# B&R Automation Studio project SuperTrak_Distribution
Automation Studio 4.12.5.95 SP; Demo project with Standard control, Axis coupling and Anti-Sloshing; technology packages: mapp 5.20.0, mappMotion 5.20.2, mappView 5.20.0

## Configuration APC910

CPU 5PC900.TS17-00, AutomationRuntime E4.91, Build 4.1.2, Safety 0.0, Vc V4.34.2

### Task classes (Cpu.sw)
```
Cyclic#1 (cycle 800 us, tolerance 0 us):
  ST_Main <- Source.SuperTrak.ST_Main.prg
  ST_Logic <- Source.SuperTrak.ST_Logic.prg
  ST_Visu <- Source.SuperTrak.ST_Visu.prg
  AxisCtrl <- Source.Axis.AxisCtrl.prg
DataObjects: McAcpSys, Acp10sys
NcDataObjects: McDriveLog
Binaries: STComTexts, McAcpDrv, udbdef, McAcpSim, mvLoader, arflatprv, McProfGen, TCLang, TCData, arcoal, arsvcreg, iomap, asfw, Config_3, Role, ashwac, sysconf, Config_2, arconfig, Config_1, TC, ashwd, Config, User, acp10cfg, Acp10map1, Acp10map, AxisConfig, OpcUaMap
Libraries: operator, AsBrMath, asstring, MpAlarmX, MpServer, McBase, MpBase, McAxis, McPureVAx, MpAxis, McAcpPar, HmiSupport, runtime, astime, AsIecCon, AsBrStr, standard, ArEventLog, AsArLog, sys_lib, McAcpAx, AsTCP, FileIO, AsIOTime, AsUDP, AsETH, AsARCfg, brsystem, AsGuard, AsHttp, AsXml, AsIOAcc, AsArSdm, AsIODiag, AsIO, AsIOMMan, DataObj, AsArProf, SuperTrak, aspciext, arssl, powerlnk, asepl, aruser, DevDetect, LogHelper, StCom
```

### Hardware
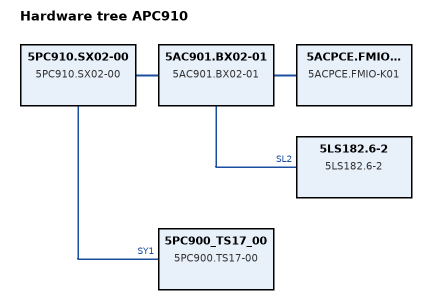
```
5AC901.BX02-01 : 5AC901.BX02-01 v1.1.1.0  [SY -> 5PC910.SX02-00.SY3]
5ACPCE.FMIO-K01 : 5ACPCE.FMIO-K01 v1.0.6.0  [SL -> 5AC901.BX02-01.SL1]
5LS182.6-2 : 5LS182.6-2 v1.9.0.0  [SL -> 5AC901.BX02-01.SL2]
  Connector IF1:
    DNAConfiguration = manual
    CycleTime = 800
5PC900_TS17_00 : 5PC900.TS17-00 v2.1.0.0  [SY -> 5PC910.SX02-00.SY1]
  ConfigurationID = SuperTrak_DistributionPackage
  UserPartitionSize = 100
  Simulation = 1
  VolatileGlobalPvSize = 262144
  TimerDeviceType = EPLX2X
  TimerDevice = 5LS182.6-2.IF1
  TaskClassIdleTime = 800
  Cyclic1Duration = 800
  Cyclic1Tolerance = 0
  Cyclic1Stack = 819600
  Cyclic2Duration = 1600
  Cyclic2Tolerance = 0
  Cyclic2Stack = 819600
  Cyclic3Duration = 49600
  Cyclic3Tolerance = 49600
  Cyclic8Duration = 9600
  FileDevice1
  FileDeviceName1 = CFast
  FileDevicePath1 = F:\
  FileDevice2
  FileDeviceName2 = Sim
  FileDevicePath2 = C:\Temp
  FtpUser1
  FtpUsername1 = Admin
  FtpUserPassword1 = TIv2O2yVOA+2iNVYi/z67sz2CqmqKSTNhuHGbiq/8uA=
  FtpUserSalt1 = e09zl50J
  FTPAccessRight1 = 0
  ActivateOpcUa = 1
  OpcUaInformationModels_PV_Version = 1
5PC910.SX02-00 : 5PC910.SX02-00 v2.1.0.0
  Connector IF1:
    AssignedOperatingSystem = ARemb
  Connector IF3:
    ActivateDevice = 1
    Mode = Manual
    InternetAddress = 192.168.13.3
    SubnetMask = 255.255.255.0
  Connector IF4:
    ActivateDevice = 1
  Connector IF5:
    AssignedOperatingSystem = ARemb
  Connector IF6:
    AssignedOperatingSystem = ARemb
  Connector IF7:
    AssignedOperatingSystem = ARemb
  Connector IF8:
    AssignedOperatingSystem = ARemb
  Connector IF9:
    AssignedOperatingSystem = ARemb
```

### Config_2.purevaxcfg - 5PC900_TS17_00/mappMotion/Config_2.purevaxcfg
```
Element PureVAxCfg_1 (Type=purevaxcfg)
  TypeID = PureVAxConfig
  PureVAxis:
    AxisReference = gAxis1
    Homing:
      Mode = Direct
        Position = 0.0
    JerkFilter = NotUsed
```

### Config_3.axis - 5PC900_TS17_00/mappMotion/Config_3.axis
```
Element gAxis1 (Type=axis)
  BaseTypeIsReadOnly = 0
  BaseType = LinearPeriodic
    MeasurementUnit = 5066068
    MeasurementResolutionIsReadOnly = 0
    MeasurementResolution = 0.01
    CountDirectionIsReadOnly = 0
    CountDirection = Standard
    PeriodSettings:
      Period = 4060
  MovementLimitsIsReadOnly = 0
  MovementLimits = Internal
    Position:
      LowerLimitMin = -1.79769313486231E308
      UpperLimitMax = 1.79769313486231E308
      LowerLimit = -1000.0
      UpperLimit = 1000.0
    VelocityIsReadOnly = 0
    Velocity:
      VelocityMax = 3.4E38
      Velocity = 4000
    AccelerationIsReadOnly = 0
    Acceleration:
      AccelerationMax = 3.4E38
      Acceleration = 10000
    DecelerationIsReadOnly = 0
    Deceleration:
      DecelerationMax = 3.4E38
      Deceleration = 10000
  Alarms = MpAlarmX
```

### Config.mpalarmxcore - 5PC900_TS17_00/mappServices/Config.mpalarmxcore
```
Element gAlarmXCore (Type=mpalarmxcore)
  mapp.AlarmX.Core.Configuration:
    [0]:
      Name = 0
      Message = Motor supply voltage out of range
      Behavior = PersistentAlarm
    [1]:
      Name = 4
      Message = Excessive coil current
      Behavior = PersistentAlarm
    [2]:
      Name = 5
      Message = High Temperature
      Behavior = PersistentAlarm
    [3]:
      Name = 7
      Message = Gateway network error
      Behavior = PersistentAlarm
    [4]:
      Name = 8
      Message = Excessive coil current (I²T)
      Behavior = PersistentAlarm
    [5]:
      Name = 9
      Message = Coil(s) unresponsive; check connections
      Behavior = PersistentAlarm
    [6]:
      Name = 11
      Message = Coil driver(s) shut down
      Behavior = PersistentAlarm
    [7]:
      Name = 14
      Message = Encoder calibration required
      Behavior = PersistentAlarm
    [8]:
      Name = 15
      Message = Excessive pallet following error
      Behavior = PersistentAlarm
    [9]:
      Name = 16
      Message = Unrecognized pallet(s) detcted
      Behavior = PersistentAlarm
    [10]:
      Name = 19
      Message = Two pallets in collision deadlook
      Behavior = PersistentAlarm
    [11]:
      Name = 20
      Message = Pallet lost position feedback
      Behavior = PersistentAlarm
    [12]:
      Name = 21
      Message = Encoder read error
      Behavior = PersistentAlarm
    [13]:
      Name = 22
      Message = Coil driver error
      Behavior = PersistentAlarm
    [14]:
      Name = 23
      Message = Conflicting pallets detected
      Behavior = PersistentAlarm
    [15]:
      Name = 24
      Message = PLC interface heartbeat timeout
      Behavior = PersistentAlarm
    [16]:
      Name = 25
      Message = Encoder communication error
      Behavior = PersistentAlarm
    [17]:
      Name = 26
      Message = Disabled pallet arrived
      Behavior = PersistentAlarm
    [18]:
      Name = 27
      Message = Abnormal condition detected
      Behavior = PersistentAlarm
    [19]:
      Name = 28
      Message = Section disabled through configuration software
      Behavior = PersistentAlarm
    [20]:
      Name = 30
      Message = Hardware initialization error
      Behavior = PersistentAlarm
    [21]:
      Name = 31
      Message = Fatal abnormal condition detected
      Behavior = PersistentAlarm
    [22]:
      Name = w0
      Message = Application warning
    [23]:
      Name = w2
      Message = License not present
    [24]:
      Name = w4
      Message = Thermal sensor malfunction
    [25]:
      Name = w5
      Message = High Temperature
    [26]:
      Name = w6
      Message = Pallet position is uncertain at destination
    [27]:
      Name = w7
      Message = Gateway network warning
    [28]:
      Name = w8
      Message = Excessive coil current (I²T)
    [29]:
      Name = w11
      Message = Pallet position correction was required
    [30]:
      Name = w12
      Message = Palled ID tag warning
    [31]:
      Name = w13
      Message = Dublicate pallet ID detected
    [32]:
      Name = w14
      Message = Two pallets in collision deadlock
    [33]:
      Name = w15
      Message = Counts out of range during Encoder handoff
    [34]:
      Name = w16
      Message = Consecutive encoder readings out of range
    [35]:
      Name = w17
      Message = Invalid region config
    [36]:
      Name = w18
      Message = Invalid parameter config
    [37]:
      Name = w19
      Message = Command failed
    [38]:
      Name = w20
      Message = Invalid syncronization zone configuration
    [39]:
      Name = w21
      Message = Encoder read warning
    [40]:
      Name = w22
      Message = Coil driver warning
    [41]:
      Name = w23
      Message = Parameter save required
    [42]:
      Name = w24
      Message = Pallet destination updated
    [43]:
      Name = w25
      Message = Encoder communication warning
    [44]:
      Name = w26
      Message = Disabled pallet arrived
    [45]:
      Name = w27
      Message = Too many pallets
    [46]:
      Name = w28
      Message = Reset required to activate configuration changes
    [47]:
      Name = w29
      Message = Excessive pallet settling time
    [48]:
      Name = w30
      Message = Controller health warning
    [49]:
      Name = w31
      Message = Abnormal condition detected
    [50]:
      Name = st0
      Message = Motor supply voltage out of range
      Behavior = PersistentAlarm
    [51]:
      Name = st4
      Message = Excessive coil current
      Behavior = PersistentAlarm
    [52]:
      Name = st5
      Message = High Temperature
      Behavior = PersistentAlarm
    [53]:
      Name = st7
      Message = Gateway network error
      Behavior = PersistentAlarm
    [54]:
      Name = st8
      Message = Excessive coil current (I²T)
      Behavior = PersistentAlarm
    [55]:
      Name = st9
      Message = Coil(s) unresponsive; check connections
      Behavior = PersistentAlarm
    [56]:
      Name = st11
      Message = Coil driver(s) shut down
      Behavior = PersistentAlarm
    [57]:
      Name = st14
      Message = Encoder calibration required
      Behavior = PersistentAlarm
    [58]:
      Name = st15
      Message = Excessive pallet following error
      Behavior = PersistentAlarm
    [59]:
      Name = st16
      Message = Unrecognized pallet(s) detcted
      Behavior = PersistentAlarm
    [60]:
      Name = st19
      Message = Two pallets in collision deadlook
      Behavior = PersistentAlarm
    [61]:
      Name = st20
      Message = Pallet lost position feedback
      Behavior = PersistentAlarm
    [62]:
      Name = st21
      Message = Encoder read error
      Behavior = PersistentAlarm
    [63]:
      Name = st22
      Message = Coil driver error
      Behavior = PersistentAlarm
    [64]:
      Name = st23
      Message = Conflicting pallets detected
      Behavior = PersistentAlarm
    [65]:
      Name = st24
      Message = PLC interface heartbeat timeout
      Behavior = PersistentAlarm
    [66]:
      Name = st25
      Message = Encoder communication error
      Behavior = PersistentAlarm
    [67]:
      Name = st26
      Message = Disabled pallet arrived
      Behavior = PersistentAlarm
    [68]:
      Name = st27
      Message = Abnormal condition detected
      Behavior = PersistentAlarm
    [69]:
      Name = st28
      Message = Section disabled through configuration software
      Behavior = PersistentAlarm
    [70]:
      Name = st30
      Message = Hardware initialization error
      Behavior = PersistentAlarm
    [71]:
      Name = st31
      Message = Fatal abnormal condition detected
      Behavior = PersistentAlarm
    [72]:
      Name = stw0
      Message = Application warning
    [73]:
      Name = stw4
      Message = Thermal sensor malfunction
    [74]:
      Name = stw5
      Message = High Temperature
    [75]:
      Name = stw7
      Message = Gateway network warning
    [76]:
      Name = stw8
      Message = Excessive coil current (I²T)
    [77]:
      Name = stw11
      Message = Pallet position correction was required
    [78]:
      Name = stw12
      Message = Palled ID tag warning
    [79]:
      Name = stw13
      Message = Dublicate pallet ID detected
    [80]:
      Name = stw15
      Message = Counts out of range during Encoder handoff
    [81]:
      Name = stw16
      Message = Consecutive encoder readings out of range
    [82]:
      Name = stw17
      Message = Invalid region config
    [83]:
      Name = stw18
      Message = Invalid parameter config
    [84]:
      Name = stw19
      Message = Command failed
    [85]:
      Name = stw20
      Message = Invalid syncronization zone configuration
    [86]:
      Name = stw21
      Message = Encoder read warning
    [87]:
      Name = stw22
      Message = Coil driver warning
    [88]:
      Name = stw23
      Message = Parameter save required
    [89]:
      Name = stw24
      Message = Pallet destination updated
    [90]:
      Name = stw25
      Message = Encoder communication warning
    [91]:
      Name = stw26
      Message = Disabled pallet arrived
    [92]:
      Name = stw27
      Message = Too many pallets
    [93]:
      Name = stw28
      Message = Reset required to active configuration changes
    [94]:
      Name = stw29
      Message = Excessive pallet settling time
    [95]:
      Name = stw30
      Message = Controller health warning
    [96]:
      Name = stw31
      Message = Abnormal condition detected
```

### Config_1.mpalarmxhistory - 5PC900_TS17_00/mappServices/Config_1.mpalarmxhistory
```
Element gAlarmXHistory (Type=mpalarmxhistory)
```

## Logical view

Binary libraries used (declarations not repeated): operator, runtime, astime, AsIecCon, AsBrStr, standard, ArEventLog, AsArLog, sys_lib, AsTCP, FileIO, AsIOTime, AsUDP, AsETH, AsARCfg, brsystem, AsGuard, AsBrMath, asstring, AsHttp, AsXml, AsIOAcc, AsArSdm, AsIODiag, AsIO, AsIOMMan, DataObj, MpBase, MpAlarmX 5.20.0, MpServer 5.20.0, AsArProf, SuperTrak 0.48.0, StCom 5.07.0, McBase 5.20.2, MpAxis 5.20.2, McPureVAx 5.20.2, McAcpPar 5.20.2, McAcpAx 5.20.2, McAxis 5.20.2

### Global.var - Global variables
```iecst
(************************************************************************************************************************************)
(************************************************************************************************************************************)
(*Global variable for internal use*)
VAR
	gStLink : {REDUND_UNREPLICABLE} StLinkType := (0); (*StCom library communication variable*)
END_VAR
(************************************************************************************************************************************)
(************************************************************************************************************************************)
(*Global variables for communication to/from SuperTrak*)
VAR
	gStCyclicControlData : {REDUND_UNREPLICABLE} ARRAY[0..499] OF USINT := [500(0)]; (*Cyclic control buffer (to SuperTrak)*)
	gStCyclicStatusData : {REDUND_UNREPLICABLE} ARRAY[0..499] OF USINT := [500(0)]; (*Cyclic status buffer (from SuperTrak)*)
	gStServiceChannelReqData : {REDUND_UNREPLICABLE} ARRAY[0..127] OF USINT := [128(0)]; (*Service channel request buffer (to SuperTrak)*)
	gStServiceChannelResData : {REDUND_UNREPLICABLE} ARRAY[0..127] OF USINT := [128(0)]; (*Service channel response buffer (from SuperTrak)*)
END_VAR
(*Variables for axis handling*)
VAR
	gMpAxisBasic_0 : MpAxisBasic; (*MpAxisBasic FUB for controlling the axis*)
	gMpAxisBasicParam : MpAxisBasicParType; (*Parameter for MpAxisBasic*)
END_VAR
(*Global status*)
VAR
	gAllSectionsEnabled : BOOL; (*Global status for SuperTrak enabled and ready*)
END_VAR
```

### Package Logical/Libraries - Global libraries

### Library Logical/Libraries/HmiSupport (IEC, version 5.06.0) - Read and write ParID from visualization
Depends on: SuperTrak, AsBrStr, ArEventLog, standard, AsIecCon, runtime

#### Types.typ - Exported data types
```iecst
(*********************************************************************************************************************************************************)
(*********************************************************************************************************************************************************)

TYPE
	HMILinkType : {REDUND_UNREPLICABLE} 	STRUCT  (*Hmi link*)
		SuperTrakStatus : {REDUND_UNREPLICABLE} HMILinkSuperTrakStatusType; (*Hmi link status*)
		LibraryStatus : {REDUND_UNREPLICABLE} HMILinkLibStatusType; (*Hmi link library status*)
	END_STRUCT;
	HMILinkSuperTrakStatusType : {REDUND_UNREPLICABLE} 	STRUCT  (*Hmi link status*)
		StatusValid : {REDUND_UNREPLICABLE} BOOL; (*Indicates if the status information is valid*)
	END_STRUCT;
	HMILinkLibStatusType : {REDUND_UNREPLICABLE} 	STRUCT  (*Hmi link library status*)
		LogBookIdent : {REDUND_UNREPLICABLE} ArEventLogIdentType; (*Ident of log book*)
		FbID : {REDUND_UNREPLICABLE} ARRAY[0..HMI_CONFIG_FBS_MINUS_ONE]OF UINT; (*Funtion block IDs*)
	END_STRUCT;
END_TYPE

(*********************************************************************************************************************************************************)
(*********************************************************************************************************************************************************)

TYPE
	HMIControlInfoType : {REDUND_UNREPLICABLE} 	STRUCT  (*Function block info*)
		Library : {REDUND_UNREPLICABLE} HMIControlLibraryType; (*Library information*)
	END_STRUCT;
	HMIControlLibraryType : {REDUND_UNREPLICABLE} 	STRUCT  (*Library information*)
		Version : {REDUND_UNREPLICABLE} STRING[8] := 'V1.0.0'; (*Actual library version*)
	END_STRUCT;
	HMIControlInternalType : {REDUND_UNREPLICABLE} 	STRUCT  (*Internal variables*)
		Step : {REDUND_UNREPLICABLE} HMIControlStepEnum; (*Step of state-machine*)
		Index : {REDUND_UNREPLICABLE} UDINT; (*Index variable*)
		Index2 : {REDUND_UNREPLICABLE} UDINT; (*Index variable*)
		Status : {REDUND_UNREPLICABLE} HMIControlInternalStatusType; (*Internal status*)
		AddErrorInfo : {REDUND_UNREPLICABLE} STRING[HMI_CONFIG_SIZE_OF_LOG_DATA]; (*Additional error information*)
		LastLogEntryID : {REDUND_UNREPLICABLE} ArEventLogRecordIDType; (*ID of last logger entry*)
		ArEventLogCreate : {REDUND_UNREPLICABLE} ArEventLogCreate; (*Function block to create log book*)
		ArEventLogGetIdent : {REDUND_UNREPLICABLE} ArEventLogGetIdent; (*Function block to get log book ident*)
		ArEventLogWrite : {REDUND_UNREPLICABLE} ArEventLogWrite; (*Function block to write log book entry*)
		CommunicationWatchdog : {REDUND_UNREPLICABLE} TON; (*Timer for communication check*)
		ErrorResetOld : {REDUND_UNREPLICABLE} BOOL; (*Marker for edge detection*)
		UpdateOld : {REDUND_UNREPLICABLE} BOOL; (*Marker for edge detection*)
	END_STRUCT;
	HMIControlInternalStatusType : {REDUND_UNREPLICABLE} 	STRUCT  (*Internal status*)
		InitConfigCheckDone : {REDUND_UNREPLICABLE} BOOL; (*Check of function block configuration done*)
		LogBookCreated : {REDUND_UNREPLICABLE} BOOL; (*Lob book created*)
		FuncitonBlockRegistered : {REDUND_UNREPLICABLE} BOOL; (*Function block registered*)
		FuncitonBlockID : {REDUND_UNREPLICABLE} UINT; (*Function block ID*)
	END_STRUCT;
END_TYPE

(*********************************************************************************************************************************************************)
(*********************************************************************************************************************************************************)

TYPE
	HMIReadParType : {REDUND_UNREPLICABLE} 	STRUCT  (*Function block parameter*)
		ParameterNumber : {REDUND_UNREPLICABLE} UINT; (*Parameter number (parameter ID) to be read*)
		SectionID : {REDUND_UNREPLICABLE} USINT; (*Section ID for paramters which are section specific*)
		StartParameterIndex : {REDUND_UNREPLICABLE} UDINT; (*Start Index of array to be read from (only for arrays)*)
		ParameterValueCount : {REDUND_UNREPLICABLE} UINT; (*Number of values (array entries) to be read after the start index (only for arrays)*)
		STRINGsize : {REDUND_UNREPLICABLE} UINT; (*Size of the string that should be read*)
	END_STRUCT;
	HMIReadInfoType : {REDUND_UNREPLICABLE} 	STRUCT  (*Function block info*)
		ErrorCode : {REDUND_UNREPLICABLE} UINT; (*Code to get the correct message*)
	END_STRUCT;
	HMIReadInternalType : {REDUND_UNREPLICABLE} 	STRUCT  (*Internal variables*)
		Step : {REDUND_UNREPLICABLE} HMIReadStepEnum; (*Step of state-machine*)
		ParametersUsed : {REDUND_UNREPLICABLE} HMIReadParType; (*Internally used parameters*)
		Index : {REDUND_UNREPLICABLE} UDINT; (*Index variable*)
		Status : {REDUND_UNREPLICABLE} HMIReadInternalStatusType; (*Internal status*)
		AddErrorInfo : {REDUND_UNREPLICABLE} STRING[HMI_CONFIG_SIZE_OF_LOG_DATA]; (*Additional error information*)
		ArEventLogWrite : {REDUND_UNREPLICABLE} ArEventLogWrite; (*Function block to write log book entry*)
		ErrorResetOld : {REDUND_UNREPLICABLE} BOOL; (*Marker for edge detection*)
		UpdateOld : {REDUND_UNREPLICABLE} BOOL; (*Marker for edge detection*)
	END_STRUCT;
	HMIReadInternalStatusType : {REDUND_UNREPLICABLE} 	STRUCT  (*Internal status*)
		InitConfigCheckDone : {REDUND_UNREPLICABLE} BOOL; (*Check of function block configuration done*)
		FuncitonBlockRegistered : {REDUND_UNREPLICABLE} BOOL; (*Function block registered*)
		FuncitonBlockID : {REDUND_UNREPLICABLE} UINT; (*Function block ID*)
		FunctionBlockIDIndex : {REDUND_UNREPLICABLE} UINT; (*Index of function block id entry*)
		InitParCheckDone : {REDUND_UNREPLICABLE} BOOL; (*Check of parameters done*)
		CommActive : {REDUND_UNREPLICABLE} BOOL; (*Indicates that service channel is occupied by this FB instance*)
		ReadStatus : {REDUND_UNREPLICABLE} UINT; (*Status of the read command*)
	END_STRUCT;
END_TYPE

(*********************************************************************************************************************************************************)
(*********************************************************************************************************************************************************)

TYPE
	HMIWriteParType : {REDUND_UNREPLICABLE} 	STRUCT  (*Function block parameter*)
		ParameterNumber : {REDUND_UNREPLICABLE} UINT; (*Parameter number (parameter ID) to be written*)
		SectionID : {REDUND_UNREPLICABLE} USINT; (*Section ID for paramters which are section specific*)
		StartParameterIndex : {REDUND_UNREPLICABLE} UDINT; (*Start Index of array to be written to (only for arrays)*)
		ParameterValueCount : {REDUND_UNREPLICABLE} UINT; (*Number of values (array entries) to be written after the start index (only for arrays)*)
		UDINTvalue : {REDUND_UNREPLICABLE} UDINT; (*UDINT variable*)
		UINTvalue : {REDUND_UNREPLICABLE} UINT; (*UINT variable*)
		USINTvalue : {REDUND_UNREPLICABLE} USINT; (*USINT variable*)
		DINTvalue : {REDUND_UNREPLICABLE} DINT; (*DINT variable*)
		INTvalue : {REDUND_UNREPLICABLE} INT; (*INT variable*)
		SINTvalue : {REDUND_UNREPLICABLE} SINT; (*SINT variable*)
		REALvalue : {REDUND_UNREPLICABLE} REAL; (*REAL variable*)
		STRINGvalue : {REDUND_UNREPLICABLE} STRING[80]; (*STRING variable*)
		STRINGsize : {REDUND_UNREPLICABLE} UINT; (*STRING size*)
		Save : {REDUND_UNREPLICABLE} HMIWriteSaveType; (*Save variable*)
	END_STRUCT;
	HMIWriteSaveType : {REDUND_UNREPLICABLE} 	STRUCT  (*Parameter save*)
		SystemLayout : {REDUND_UNREPLICABLE} BOOL; (*Save system layout*)
		Targets : {REDUND_UNREPLICABLE} BOOL; (*Save targets*)
		Regions : {REDUND_UNREPLICABLE} BOOL; (*Save regions*)
		MoveConfig : {REDUND_UNREPLICABLE} BOOL; (*Save move configuration*)
		GlobalPar : {REDUND_UNREPLICABLE} BOOL; (*Save global parameters*)
		Offsets : {REDUND_UNREPLICABLE} BOOL; (*Save offsets*)
		SectionPar : {REDUND_UNREPLICABLE} BOOL; (*Save section parameters*)
		ControlGains : {REDUND_UNREPLICABLE} BOOL; (*Save control gains*)
		EncoderConfig : {REDUND_UNREPLICABLE} BOOL; (*Save encoder calibration and configuration*)
		IRTagConfig : {REDUND_UNREPLICABLE} BOOL; (*Save IR tag configuration*)
		VirtualIO : {REDUND_UNREPLICABLE} BOOL; (*Save virtual IOs*)
		PosTrig : {REDUND_UNREPLICABLE} BOOL; (*Save position triggers*)
	END_STRUCT;
	HMIWriteInfoType : {REDUND_UNREPLICABLE} 	STRUCT  (*Function block info*)
		ErrorCode : {REDUND_UNREPLICABLE} UINT; (*Code to get the correct message*)
	END_STRUCT;
	HMIWriteInternalType : {REDUND_UNREPLICABLE} 	STRUCT  (*Internal variables*)
		Step : {REDUND_UNREPLICABLE} HMIWriteStepEnum; (*Step of state-machine*)
		ParametersUsed : {REDUND_UNREPLICABLE} HMIWriteParType; (*Internally used parameters*)
		Index : {REDUND_UNREPLICABLE} UDINT; (*Index variable*)
		Status : {REDUND_UNREPLICABLE} HMIWriteInternalStatusType; (*Internal status*)
		AddErrorInfo : {REDUND_UNREPLICABLE} STRING[HMI_CONFIG_SIZE_OF_LOG_DATA]; (*Additional error information*)
		ArEventLogWrite : {REDUND_UNREPLICABLE} ArEventLogWrite; (*Function block to write log book entry*)
		ErrorResetOld : {REDUND_UNREPLICABLE} BOOL; (*Marker for edge detection*)
		UpdateOld : {REDUND_UNREPLICABLE} BOOL; (*Marker for edge detection*)
		SaveValue : {REDUND_UNREPLICABLE} UDINT; (*Parameter that should be saved*)
	END_STRUCT;
	HMIWriteInternalStatusType : {REDUND_UNREPLICABLE} 	STRUCT  (*Internal status*)
		InitConfigCheckDone : {REDUND_UNREPLICABLE} BOOL; (*Check of function block configuration done*)
		FuncitonBlockRegistered : {REDUND_UNREPLICABLE} BOOL; (*Function block registered*)
		FuncitonBlockID : {REDUND_UNREPLICABLE} UINT; (*Function block ID*)
		FunctionBlockIDIndex : {REDUND_UNREPLICABLE} UINT; (*Index of function block id entry*)
		InitParCheckDone : {REDUND_UNREPLICABLE} BOOL; (*Check of parameters done*)
		CommActive : {REDUND_UNREPLICABLE} BOOL; (*Indicates that service channel is occupied by this FB instance*)
		WriteStatus : {REDUND_UNREPLICABLE} UINT; (*Internal status of the write command*)
	END_STRUCT;
END_TYPE

(*********************************************************************************************************************************************************)
(*********************************************************************************************************************************************************)

TYPE
	HMIControlStepEnum :
		( (*Steps for state-machine*)
		HMI_CTRL_STATE_INIT := 0, (*Init state*)
		HMI_CTRL_STATE_INIT_CHECK_CONFIG := 1, (*Check configuration*)
		HMI_CTRL_STATE_CREATE_LOGBOOK := 2, (*Create Logbook*)
		HMI_CTRL_STATE_REGISTER_FB := 3, (*Register FUB*)
		HMI_CTRL_STATE_OPERATION := 10, (*Operation*)
		HMI_CTRL_STATE_ERROR := 255 (*Error*)
		);
	HMIWriteStepEnum :
		( (*Steps for state-machine*)
		HMI_WPAR_STATE_INIT := 0, (*Init state*)
		HMI_WPAR_STATE_INIT_CHECK_CONFIG := 1, (*Check configuration*)
		HMI_WPAR_STATE_INIT_REG_FB := 2, (*Register FUB*)
		HMI_WPAR_STATE_INIT_CHECK_PAR := 3, (*Check parameter*)
		HMI_WPAR_STATE_OPERATION := 10, (*Operation*)
		HMI_WPAR_STATE_ERROR := 255 (*Error*)
		);
	HMIReadStepEnum :
		( (*Steps for state-machine*)
		HMI_RPAR_STATE_INIT := 0, (*Init state*)
		HMI_RPAR_STATE_INIT_CHECK_CONFIG := 1, (*Check configuration*)
		HMI_RPAR_STATE_INIT_REG_FB := 2, (*Register FUB*)
		HMI_RPAR_STATE_INIT_CHECK_PAR := 3, (*Check parameter*)
		HMI_RPAR_STATE_OPERATION := 10, (*Operation*)
		HMI_RPAR_STATE_ERROR := 255 (*Error*)
		);
END_TYPE
```

#### Constants.var - Exported constants
```iecst
(********************************************************************************************************************************************************************************************************************************************)
(********************************************************************************************************************************************************************************************************************************************)
(*Configuration*)
VAR CONSTANT
	HMI_CONFIG_VERSION : STRING[8] := 'V5.6.0'; (*Library version*)
	HMI_CONFIG_SIZE_OF_LOG_DATA : USINT := 250; (*Size of additional information in log book entry (in bytes)*)
	HMI_CONFIG_FB_ID_HMICONTROL : UINT := 2#0001000000000000; (*Function block type ID for HMIControl*)
	HMI_CONFIG_FB_ID_HMIREAD : UINT := 2#0010000000000000; (*Function block type ID for HMIRead*)
	HMI_CONFIG_FB_ID_HMIWRITE : UINT := 2#0011000000000000; (*Function block type ID for HMIWrite*)
	HMI_CONFIG_NR_OF_SECTIONS : USINT := 64; (*Max number of sections*)
	HMI_CONFIG_MAX_NR_OF_FBS : UINT := 1024; (*Max number of function blocks*)
	HMI_CONFIG_COMM_TIME_OUT : TIME := T#500ms; (*Communication time out limit*)
	HMI_CONFIG_SERV_CH_TASK_READ : USINT := 5; (*Command ID to read paramter through service channel*)
	HMI_CONFIG_SERV_CH_TASK_WRITE : USINT := 6; (*Command ID to write paramter through service channel*)
	HMI_CONFIG_SERV_CH_MAX_DATA : USINT := 32; (*Maxumum size of data response from service channel in bytes*)
	HMI_CONFIG_CMD_IF_BYTE_STRUCT : USINT := 4; (*The communication interface has to be aligned to 4 bytes*)
	HMI_SC_CODE_SUCCESS : USINT := 0; (*Response from SuperTrak that message is OK*)
	HMI_SC_CODE_WRONG_SECTION_ID : USINT := 1; (*Response from SuperTrak that section ID is invalid*)
	HMI_SC_CODE_WRONG_PAR_ID : USINT := 2; (*Response from SuperTrak that paramter ID is invalid*)
	HMI_SC_CODE_WRONG_TASK : USINT := 3; (*Response from SuperTrak that task is invalid*)
	HMI_SC_CODE_TASK_UNAVAILABLE : USINT := 4; (*Response from SuperTrak that task is currently unavailable*)
	HMI_SC_CODE_WRONG_PAR_IDX : USINT := 6; (*Response from SuperTrak that start index is invalid*)
	HMI_SC_CODE_WRONG_PAR_VALUE : USINT := 7; (*Response from SuperTrak that paramter value is invalid*)
	HMI_SC_CODE_WRONG_PAR_COUNT : USINT := 8; (*Response from SuperTrak that paramter count is invalid*)
	HMI_SC_CODE_TIMEOUT : USINT := 10; (*Response from SuperTrak that Communication timed out*)
	HMI_SC_CODE_NOT_AUTHORIZED : USINT := 13; (*Response from SuperTrak that access is not authorized*)
	HMI_SC_CODE_INVALID_PACKET : USINT := 14; (*Response from SuperTrak that packet is invalid*)
	HMI_SC_CODE_INTERNAL_ERROR : USINT := 15; (*Response from SuperTrak that internal error occured*)
	HMI_SC_SAVE_PARAMTER_CODE : UINT := 971; (*PNU to save parameters*)
	HMI_SC_SAVE_PARAMTER_CMD : UDINT := 60028; (*Bitwise parameter save HMImands (see TrakMaster help for more information)*)
	HMI_PNU_SECTION_COUNT : UINT := 1080; (*Parameter ID for section count*)
	HMI_PNU_SYSTEM_NAME : UINT := 1053; (*Parameter ID for system name*)
	HMI_PNU_ENABLE_CONTROL : UINT := 1057; (*Parameter ID for enable control*)
	HMI_PNU_CMD_IF_SECTIONS : UINT := 1432; (*Parameter ID for section count in Command interface*)
	HMI_PNU_CMD_IF_TARGETS : UINT := 1434; (*Parameter ID for target count in Command interface*)
	HMI_PNU_CMD_IF_COMMANDS : UINT := 1436; (*Parameter ID for Command count in Command interface*)
	HMI_PNU_CMD_IF_OPTIONS : UINT := 1430; (*Parameter ID for Command interface options*)
END_VAR
(**)
(********************************************************************************************************************************************************************************************************************************************)
(********************************************************************************************************************************************************************************************************************************************)
(*Derivated Constants*)
VAR CONSTANT
	HMI_CONFIG_SECTIONS_MINUS_ONE : USINT := HMI_CONFIG_NR_OF_SECTIONS-1; (*Derivated constant*)
	HMI_CONFIG_FBS_MINUS_ONE : UINT := HMI_CONFIG_MAX_NR_OF_FBS-1; (*Derivated constant*)
	HMI_CONFIG_SERV_CH_MAX_DATA_M1 : USINT := HMI_CONFIG_SERV_CH_MAX_DATA-1; (*Derivated constant*)
END_VAR
(**)
(********************************************************************************************************************************************************************************************************************************************)
(********************************************************************************************************************************************************************************************************************************************)
(*Error-Code, Warning-Code, Information-Code, Success-Code*)
VAR CONSTANT
	HMI_NO_ERROR : DINT := 0; (*No error, warning, information etc. present*)
	HMI_ERR_FB_INSTANCE_REG : DINT := -536805375; (*Instance of this function block already registered*)
	HMI_ERR_WRONG_PARAMETER : DINT := -536805373; (*Wrong parameter*)
	HMI_ERR_COMMUNICAITON_TIME_OUT : DINT := -536805372; (*Timeout for Communication to SuperTrak*)
	HMI_ERR_NO_HMICONTROL_REG : DINT := -536805371; (*There is no instance of HMIControl registered*)
	HMI_ERR_SUPERTRAK_SYS : DINT := -536805370; (*SuperTrak reported an system error*)
	HMI_ERR_WRONG_CONFIG : DINT := -536805369; (*Address not valid, or Target/Section/ShuttleID not vaild*)
	HMI_ERR_CMD_NOT_EXECUTED : DINT := -536805368; (*Command could not be executed successfully*)
	HMI_ERR_SUPERTRAK_SEC : DINT := -536805367; (*SuperTrak reported an section error*)
	HMI_ERR_SERVICE_CHANNEL_FAULT : DINT := -536805366; (*SuperTrak responded with an error to a service channel request*)
	HMI_ERR_CMD_HANDSHAKE : DINT := -536805365; (*CommandComplete flag is true before Command execution*)
	HMI_WRN_SUPERTRAK_SYS : DINT := -1610547099; (*SuperTrak reported a system warning*)
	HMI_WRN_SUPERTRAK_SEC : DINT := -1610547098; (*SuperTrak reported a section warning*)
	HMI_WRN_ENABLE_SIGNAL_SOURCE : DINT := -1610547097; (*Enable signal source configuration doesn't allow this Command*)
	HMI_INFO_COMM_STRUCT_TOO_BIG : DINT := 1610678473; (*The Communication structure is too big*)
	HMI_SUCC_FB_REGISTRATION : DINT := 536936749; (*The function block was registered successfully*)
	HMI_SUCC_PARAM_VALID : DINT := 536936750; (*Parameters valid*)
END_VAR
```

#### HmiSupport.fun - Exported functions and function blocks
```iecst
FUNCTION_BLOCK HMIControl (*This function block is used as connection between the Hmi function blocks. This funciton block also creates the logbook for this library*) (*$Group=User,$CAT=User,$GROUPICON=User.png,$CATICON=User.png*)
	VAR_INPUT
		HMILink : REFERENCE TO HMILinkType; (*Connection to other Hmi function blocks*) (* *) (*#PAR*)
		Enable : BOOL; (*Enables the function block*) (* *) (*#PAR*)
		ErrorReset : BOOL; (*Resets the function block errors*) (* *) (*#PAR*)
		Update : BOOL; (*Updates the parameters*) (* *) (*#PAR*)
	END_VAR
	VAR_OUTPUT
		Active : BOOL; (*Indicates whether the function block is active*) (* *) (*#PAR*)
		Error : BOOL; (*Indicates that the funciton block is in an error state or a command was not executed correctly*) (* *) (*#PAR*)
		StatusID : DINT; (*Status information about the function block*) (* *) (*#PAR*)
		UpdateDone : BOOL; (*Parameter update completed*) (* *) (*#PAR*)
		Info : HMIControlInfoType; (*Additional information about the library*) (* *) (*#PAR*)
	END_VAR
	VAR
		Internal : HMIControlInternalType; (*Internal variables*) (* *) (*#OMIT*)
	END_VAR
END_FUNCTION_BLOCK

FUNCTION_BLOCK HMIReadParID (*This function block can be used to read ParIDs from SuperTrak with a HMI.*) (*$Group=User,$CAT=User,$GROUPICON=User.png,$CATICON=User.png*)
	VAR_INPUT
		HMILink : REFERENCE TO HMILinkType; (*Connection to other Hmi function blocks*) (* *) (*#PAR*)
		Enable : BOOL; (*Enables the function block*) (* *) (*#PAR*)
		ErrorReset : BOOL; (*Resets function block errors*) (* *) (*#PAR*)
		Parameters : REFERENCE TO HMIReadParType; (*Function block parameters*) (* *) (*#PAR*)
		Update : BOOL; (*Updates the parameters*) (* *) (*#PAR*)
		ReadUDINT : BOOL; (*Read UDINT ParID*) (* *) (*#CMD*)
		ReadUINT : BOOL; (*Read UINT ParID*) (* *) (*#CMD*)
		ReadUSINT : BOOL; (*Read USINT ParID*) (* *) (*#CMD*)
		ReadDINT : BOOL; (*Read DINT ParID*) (* *) (*#CMD*)
		ReadINT : BOOL; (*Read INT ParID*) (* *) (*#CMD*)
		ReadSINT : BOOL; (*Read SINT ParID*) (* *) (*#CMD*)
		ReadREAL : BOOL; (*Read REAL ParID*) (* *) (*#CMD*)
		ReadSTRING : BOOL; (*Read STRING ParID*) (* *) (*#CMD*)
	END_VAR
	VAR_OUTPUT
		Active : BOOL; (*Indicates whether the function block is active*) (* *) (*#PAR*)
		Error : BOOL; (*Indicates that the function block is in an error state or a command was not executed correctly*) (* *) (*#PAR*)
		StatusID : DINT; (*Status information about the function block*) (* *) (*#PAR*)
		UpdateDone : BOOL; (*Parameter update completed*) (* *) (*#PAR*)
		Out_UDINT : UDINT; (*UDINT output*) (* *) (*#CMD*)
		Out_UINT : UINT; (*UINT output*) (* *) (*#CMD*)
		Out_USINT : USINT; (*USINT output*) (* *) (*#CMD*)
		Out_DINT : DINT; (*DINT output*) (* *) (*#CMD*)
		Out_INT : INT; (*INT output*) (* *) (*#CMD*)
		Out_SINT : SINT; (*SINT output*) (* *) (*#CMD*)
		Out_REAL : REAL; (*REAL output*) (* *) (*#CMD*)
		Out_STRING : STRING[80]; (*STRING output*) (* *) (*#CMD*)
		CommandDone : BOOL; (*Command successfully executed by the function block*) (* *) (*#CMD*)
		Info : HMIReadInfoType; (*Function block informations*) (* *) (*#PAR*)
	END_VAR
	VAR
		Internal : HMIReadInternalType; (*Internal variables*) (* *) (*#OMIT*)
	END_VAR
END_FUNCTION_BLOCK

FUNCTION_BLOCK HMIWriteParID (*This function block can be used to write ParIDs from SuperTrak with a HMI.*) (*$Group=User,$CAT=User,$GROUPICON=User.png,$CATICON=User.png*)
	VAR_INPUT
		HMILink : REFERENCE TO HMILinkType; (*Connection to other Hmi function blocks*) (* *) (*#PAR*)
		Enable : BOOL; (*Enables the function block*) (* *) (*#PAR*)
		ErrorReset : BOOL; (*Resets function block errors*) (* *) (*#PAR*)
		Parameters : REFERENCE TO HMIWriteParType; (*Function block parameters*) (* *) (*#PAR*)
		Update : BOOL; (*Updates the parameters*) (* *) (*#PAR*)
		WriteUDINT : BOOL; (*Write UDINT ParID*) (* *) (*#CMD*)
		WriteUINT : BOOL; (*Write UINT ParID*) (* *) (*#CMD*)
		WriteUSINT : BOOL; (*Write USINT ParID*) (* *) (*#CMD*)
		WriteDINT : BOOL; (*Write DINT ParID*) (* *) (*#CMD*)
		WriteINT : BOOL; (*Write INT ParID*) (* *) (*#CMD*)
		WriteSINT : BOOL; (*Write SINT ParID*) (* *) (*#CMD*)
		WriteREAL : BOOL; (*Write REAL ParID*) (* *) (*#CMD*)
		WriteSTRING : BOOL; (*Write STRING ParID*) (* *) (*#CMD*)
		SaveParameters : BOOL; (*Save parameters*) (* *) (*#CMD*)
	END_VAR
	VAR_OUTPUT
		Active : BOOL; (*Indicates whether the function block is active*) (* *) (*#PAR*)
		Error : BOOL; (*Indicates that the function block is in an error state or a command was not executed correctly*) (* *) (*#PAR*)
		StatusID : DINT; (*Status information about the function block*) (* *) (*#PAR*)
		UpdateDone : BOOL; (*Parameter update completed*) (* *) (*#PAR*)
		CommandDone : BOOL; (*Command successfully executed by the function block*) (* *) (*#CMD*)
		Info : HMIWriteInfoType; (*Function block informations*) (* *) (*#PAR*)
	END_VAR
	VAR
		Internal : HMIWriteInternalType; (*Internal variables*) (* *) (*#OMIT*)
	END_VAR
END_FUNCTION_BLOCK
```

#### HmiControl.st - HmiControl function block
```iecst
(******************************************************************************************
 * Copyright: Bernecker + Rainer
 * Author:  B+R
 * Created:  July 2, 2018/08:25 AM
 ******************************************************************************************
 ******************************************************************************************
 * Version History:
 * ----------------------------------------------------------------------------------------
 * V 1.00.0   July 2, 2018/08:25 AM  First Version
 ******************************************************************************************
 * Description:
 * ----------------------------------------------------------------------------------------
 * July 2, 2018/08:25 AM V1.00.0:
 * This function block writes error data into the logger from other FUBs of this library.
 ******************************************************************************************)

FUNCTION_BLOCK HMIControl

	// Check if function block is enabled
	IF Enable THEN
		//####################################################################################//
		// FUNCTION BLOCK IS ENABLED
		//####################################################################################//

		// Set Library version information
		Info.Library.Version															:= HMI_CONFIG_VERSION;

		// Check if error occured to change state
		IF Error THEN
			// Go to state error, to wait for acknowledge
			Internal.Step																:= HMI_CTRL_STATE_ERROR;
		END_IF;

		//************************************************************************************//
		// Operation
		//************************************************************************************//
		CASE Internal.Step OF
			//--------------------------------------------------------------------------------//
			// Initialize internal parameters
			//--------------------------------------------------------------------------------//
			HMI_CTRL_STATE_INIT:

				// Initialize function block to create a logbook
				Internal.ArEventLogCreate.Info											:= 0;	// Reserved (see AS help)
				Internal.ArEventLogCreate.Name											:= 'HMILib';
				Internal.ArEventLogCreate.Persistence									:= arEVENTLOG_PERSISTENCE_PERSIST;
				Internal.ArEventLogCreate.Size											:= 65536;

				Internal.ArEventLogGetIdent.Name										:= Internal.ArEventLogCreate.Name;

				// Initialize function block creating a logbook entry
				Internal.ArEventLogWrite.AddData										:= ADR(Internal.AddErrorInfo);
				Internal.ArEventLogWrite.AddDataFormat									:= 1;	// zero-terminated string
				Internal.ArEventLogWrite.AddDataSize									:= SIZEOF(Internal.AddErrorInfo);
				Internal.ArEventLogWrite.ObjectID										:= 'HmiControl';

				Internal.ArEventLogWrite.OriginRecordID									:= 0;	// don't use origin record
				Internal.ArEventLogWrite.TimeStamp										:= 0;	// use internal time stamp

				// Initialize communication watchdog
				Internal.CommunicationWatchdog.PT										:= HMI_CONFIG_COMM_TIME_OUT;

				Internal.Step															:= HMI_CTRL_STATE_INIT_CHECK_CONFIG;

				//--------------------------------------------------------------------------------//
				// First check of function block configuration
				//--------------------------------------------------------------------------------//
			HMI_CTRL_STATE_INIT_CHECK_CONFIG:

				// Check if given addresses are valid
				IF (ADR(HMILink) > 0) THEN

					Internal.Status.InitConfigCheckDone									:= TRUE;
					Internal.Step														:= HMI_CTRL_STATE_CREATE_LOGBOOK;
				ELSE
					Internal.Status.InitConfigCheckDone									:= FALSE;
					// Address not valid, set error
					StatusID															:= HMI_ERR_WRONG_CONFIG;
					Error																:= TRUE;
				END_IF;

				//--------------------------------------------------------------------------------//
				// Create logbook for all function blocks
				//--------------------------------------------------------------------------------//
			HMI_CTRL_STATE_CREATE_LOGBOOK:

				// Set command to create logbook
				Internal.ArEventLogCreate.Execute										:= TRUE;
				Internal.ArEventLogCreate();

				// Check if logbook is created successfully, to continue
				IF Internal.ArEventLogCreate.Done THEN
					// Reset command
					Internal.ArEventLogCreate.Execute									:= FALSE;
					Internal.Status.LogBookCreated										:= TRUE;
					// Save Ident of logbook
					Internal.ArEventLogWrite.Ident										:= Internal.ArEventLogCreate.Ident;
					HMILink.LibraryStatus.LogBookIdent									:= Internal.ArEventLogCreate.Ident;
					Internal.ArEventLogCreate();

					// Create logbook entry
					Internal.AddErrorInfo												:= 'HMI Version ';
					brsstrcat(ADR(Internal.AddErrorInfo), ADR(HMI_CONFIG_VERSION));

					Internal.ArEventLogWrite.EventID									:= HMI_SUCC_FB_REGISTRATION;
					// Write logbook entry
					WriteLogbookEntry;

					Internal.Step														:= HMI_CTRL_STATE_REGISTER_FB;

					// Check if logbook already exists, to continue
				ELSIF (Internal.ArEventLogCreate.StatusID = arEVENTLOG_ERR_LOGBOOK_EXISTS) THEN
					// Get logbook ident
					Internal.ArEventLogGetIdent.Execute									:= TRUE;
					Internal.ArEventLogGetIdent();

					// Wait until FB is done getting the ident
					IF Internal.ArEventLogGetIdent.Done THEN
						// Copy ident
						Internal.ArEventLogWrite.Ident									:= Internal.ArEventLogGetIdent.Ident;
						HMILink.LibraryStatus.LogBookIdent								:= Internal.ArEventLogGetIdent.Ident;
						// Reset command
						Internal.ArEventLogCreate.Execute								:= FALSE;
						Internal.ArEventLogGetIdent.Execute								:= FALSE;
						Internal.Status.LogBookCreated									:= TRUE;
						Internal.ArEventLogCreate();
						Internal.ArEventLogGetIdent();

						// Create logbook entry
						Internal.AddErrorInfo											:= 'HMI Version ';
						brsstrcat(ADR(Internal.AddErrorInfo), ADR(HMI_CONFIG_VERSION));

						Internal.ArEventLogWrite.EventID								:= HMI_SUCC_FB_REGISTRATION;
						// Write logbook entry
						WriteLogbookEntry;

						Internal.Step													:= HMI_CTRL_STATE_REGISTER_FB;
					END_IF;

					// If creation of logbook was not successfull, set error
				ELSIF Internal.ArEventLogCreate.Error THEN
					// Copy status id of failed funciton block
					StatusID															:= Internal.ArEventLogCreate.StatusID;
					Internal.Status.LogBookCreated										:= FALSE;
					Internal.ArEventLogCreate.Execute									:= FALSE;
					Internal.ArEventLogCreate();
					Error																:= TRUE;
				END_IF;

				//--------------------------------------------------------------------------------//
				// Register function block in HMILink structure
				//--------------------------------------------------------------------------------//
			HMI_CTRL_STATE_REGISTER_FB:

				// Build function block ID
				Internal.Status.FuncitonBlockID											:= HMI_CONFIG_FB_ID_HMICONTROL;

				// Check if FB is already registered
				IF Internal.Status.FuncitonBlockRegistered THEN
					Internal.Step														:= HMI_CTRL_STATE_OPERATION;

					// If this function block ID is not yet used and the FB is not registered, register FB, otherwise set error,
					// because there can only be one instance OF this FB
				ELSIF (HMILink.LibraryStatus.FbID[0] <> Internal.Status.FuncitonBlockID) THEN
					// For StControl, use always index 0
					HMILink.LibraryStatus.FbID[0]										:= Internal.Status.FuncitonBlockID;
					Internal.Status.FuncitonBlockRegistered								:= TRUE;

					// Create logbook entry
					Internal.AddErrorInfo												:= 'Function block registration successfull';
					Internal.ArEventLogWrite.EventID									:= HMI_SUCC_FB_REGISTRATION;
					// Write logbook entry
					WriteLogbookEntry;
					Internal.Step														:= HMI_CTRL_STATE_OPERATION;

				ELSE
					// Create logbook entry
					Internal.AddErrorInfo												:= 'Another instance of this function block is already registered';
					Internal.ArEventLogWrite.EventID									:= HMI_ERR_FB_INSTANCE_REG;
					// Write logbook entry
					WriteLogbookEntry;
					// StControl instance is already in use, set error
					StatusID															:= HMI_ERR_FB_INSTANCE_REG;
					Error																:= TRUE;
				END_IF;

				//--------------------------------------------------------------------------------//
				// Operation
				//--------------------------------------------------------------------------------//
			HMI_CTRL_STATE_OPERATION:

				// Set active output
				Active																		:= TRUE;

				IF (ADR(HMILink) > 0) THEN
					//:::::::::::::::::::::::::::::::::::::::::::::::::::::::::::::::::::::::::::://
					// Parameter update handling
					// Check if parameters should be updated
					IF Update AND NOT Internal.UpdateOld AND NOT UpdateDone THEN
						UpdateDone															:= TRUE;
					ELSIF NOT Update THEN
						UpdateDone															:= FALSE;
					END_IF;

					// Set valid
					HMILink.SuperTrakStatus.StatusValid									:= TRUE;
				END_IF;

			//--------------------------------------------------------------------------------//
			// Error handling
			//--------------------------------------------------------------------------------//
			HMI_CTRL_STATE_ERROR:

				// Reset outputs
				Active																	:= FALSE;
				UpdateDone																:= FALSE;

				// Return to previous state, if error is cleared
				IF NOT Error THEN
					// Check in which state to jump
					IF NOT Internal.Status.InitConfigCheckDone THEN
						Internal.Step													:= HMI_CTRL_STATE_INIT_CHECK_CONFIG;
					ELSIF NOT Internal.Status.LogBookCreated THEN
						Internal.Step													:= HMI_CTRL_STATE_CREATE_LOGBOOK;
					ELSIF NOT Internal.Status.FuncitonBlockRegistered THEN
						Internal.Step													:= HMI_CTRL_STATE_REGISTER_FB;
					ELSE
						Internal.Step													:= HMI_CTRL_STATE_OPERATION;
					END_IF;
				END_IF;
		END_CASE;

		//************************************************************************************//
		// Error and Warning acknowledgement
		//************************************************************************************//

		// Check if error or warning is acknowledged by user
		IF ErrorReset AND Error AND NOT Internal.ErrorResetOld THEN
			// Reset error
			StatusID																	:= HMI_NO_ERROR;
			Error																		:= FALSE;
		ELSIF ErrorReset AND StatusID <> HMI_NO_ERROR AND NOT Internal.ErrorResetOld THEN
			// Reset warning
			StatusID																	:= HMI_NO_ERROR;
		END_IF;

		Internal.ErrorResetOld															:= ErrorReset;
		Internal.UpdateOld																:= Update;

		//************************************************************************************//
		// Function block calls
		//************************************************************************************//
		Internal.CommunicationWatchdog();

	ELSE
		//####################################################################################//
		// FUNCTION BLOCK IS DISABLED
		//####################################################################################//
		// Reset all outputs
		Active																			:= FALSE;
		Error																			:= FALSE;
		StatusID																		:= HMI_NO_ERROR;
		UpdateDone																		:= FALSE;

		// Reset state machine
		Internal.Step																	:= HMI_CTRL_STATE_INIT;
		// Check if address is valid, to avoid system crash
		IF (ADR(HMILink) > 0) THEN
			// Unregister function block (if registered)
			IF Internal.Status.FuncitonBlockRegistered THEN
				HMILink.LibraryStatus.FbID[0]											:= 0;
				Internal.Status.FuncitonBlockRegistered									:= FALSE;
			END_IF;
		END_IF;

		Internal.Status.LogBookCreated													:= FALSE;
		Internal.CommunicationWatchdog.IN												:= FALSE;

	END_IF;

END_FUNCTION_BLOCK
```

#### HmiReadParID.st - HmiReadParID function block
```iecst
(******************************************************************************************
 * Copyright: Bernecker + Rainer
 * Author:  B+R
 * Created:  July 2, 2018/09:40 AM
 ******************************************************************************************
 ******************************************************************************************
 * Version History:
 * ----------------------------------------------------------------------------------------
 * V 1.00.0   July 2, 2018/09:40 AM  First Version
 ******************************************************************************************
 * Description:
 * ----------------------------------------------------------------------------------------
 * July 2, 2018/09:40 AM V1.00.0:
 * This FUNCTION block reads ParIDs from the SuperTrak.
 * The FUB can be connected directly to a HMI application.
 * The parameter structure and I/Os can be used inside the visu without extra implementation.
 ******************************************************************************************)

FUNCTION_BLOCK HMIReadParID
		// Check if function block is enabled
	IF Enable THEN
		//####################################################################################//
		// FUNCTION BLOCK IS ENABLED
		//####################################################################################//

		// Check if error occured to change state
		IF Error THEN
			// Go to state error, to wait for acknowledge
			Internal.Step																	:= HMI_RPAR_STATE_ERROR;
		END_IF;

		//************************************************************************************//
		// Operation
		//************************************************************************************//
		CASE Internal.Step OF
			//--------------------------------------------------------------------------------//
			// Initialize internal parameters
			//--------------------------------------------------------------------------------//
			HMI_RPAR_STATE_INIT:

				// Initialize function block to create a logbook entry
				Internal.ArEventLogWrite.AddData											:= ADR(Internal.AddErrorInfo);
				Internal.ArEventLogWrite.AddDataFormat										:= 1;	// zero-terminated string
				Internal.ArEventLogWrite.AddDataSize										:= SIZEOF(Internal.AddErrorInfo);
				Internal.ArEventLogWrite.ObjectID											:= 'HMIReadParID';
				Internal.AddErrorInfo														:= '';
				Internal.ArEventLogWrite.OriginRecordID										:= 0;	// don't use origin record
				Internal.ArEventLogWrite.TimeStamp											:= 0;	// use internal time stamp

				Internal.Step																:= HMI_RPAR_STATE_INIT_CHECK_CONFIG;

				//--------------------------------------------------------------------------------//
				// Register function block
				//--------------------------------------------------------------------------------//
			HMI_RPAR_STATE_INIT_CHECK_CONFIG:

				// Check configuration inputs if valid
				IF (ADR(Parameters) > 0) AND
					(ADR(HMILink) > 0) THEN
					// Config OK
					Internal.Status.InitConfigCheckDone										:= TRUE;
					Internal.Step															:= HMI_RPAR_STATE_INIT_REG_FB;
				ELSE
					Internal.Status.InitConfigCheckDone										:= FALSE;
					// Set error
					StatusID																:= HMI_ERR_WRONG_CONFIG;
					Error																	:= TRUE;
				END_IF;

				//--------------------------------------------------------------------------------//
				// Register function block
				//--------------------------------------------------------------------------------//
			HMI_RPAR_STATE_INIT_REG_FB:

				// Check if function block is not registered yet
				IF NOT Internal.Status.FuncitonBlockRegistered THEN
					// Check if StControl instance is present and valid
					IF (HMILink.LibraryStatus.FbID[0] <> 0) AND (HMILink.LibraryStatus.LogBookIdent <> 0) THEN
						// Save logbook ident
						Internal.ArEventLogWrite.Ident										:= HMILink.LibraryStatus.LogBookIdent;
						// Create function block ID
						Internal.Status.FuncitonBlockID										:= HMI_CONFIG_FB_ID_HMIREAD;
						Internal.Status.FunctionBlockIDIndex								:= 0;
						Internal.Status.FuncitonBlockRegistered								:= TRUE;
						// Create logbook entry
						Internal.AddErrorInfo												:= 'Function block registration successfull';
						Internal.ArEventLogWrite.EventID									:= HMI_SUCC_FB_REGISTRATION;
						// Write logbook entry
						WriteLogbookEntry;
					ELSIF (HMILink.LibraryStatus.LogBookIdent <> 0) THEN
						Internal.AddErrorInfo												:= 'No enabled instance of HMIControl could be found';
						Internal.ArEventLogWrite.EventID									:= HMI_ERR_NO_HMICONTROL_REG;
						// Write logbook entry
						WriteLogbookEntry;
						// Set error
						StatusID															:= HMI_ERR_NO_HMICONTROL_REG;
						Error																:= TRUE;
					ELSE
						// Set error
						StatusID															:= HMI_ERR_NO_HMICONTROL_REG;
						Error																:= TRUE;
					END_IF;
				ELSE
					// Continue
					Internal.Step															:= HMI_RPAR_STATE_INIT_CHECK_PAR;
				END_IF;

				//--------------------------------------------------------------------------------//
				// Check parameters
				//--------------------------------------------------------------------------------//
			HMI_RPAR_STATE_INIT_CHECK_PAR:

				// Save parameters
				Internal.ParametersUsed														:= Parameters;
				Internal.Status.InitParCheckDone											:= TRUE;
				Internal.Step																:= HMI_RPAR_STATE_OPERATION;

				//--------------------------------------------------------------------------------//
				// Operation
				//--------------------------------------------------------------------------------//
			HMI_RPAR_STATE_OPERATION:

				// Set active output
				Active																		:= TRUE;

				// Check configuration inputs if valid
				IF (ADR(Parameters) > 0) AND
					(ADR(HMILink) > 0) THEN
					//:::::::::::::::::::::::::::::::::::::::::::::::::::::::::::::::::::::::::::://
					// Parameter update handling
					// Check if parameters should be updated
					IF Update AND NOT Internal.UpdateOld AND NOT UpdateDone THEN

						// Check if parameters are valid
						IF (Parameters.ParameterNumber <> 0) AND
							(Parameters.SectionID <= HMI_CONFIG_NR_OF_SECTIONS) THEN
							// PARAMTERS ARE VALID
							// copy paramters to internal stucture
							Internal.ParametersUsed												:= Parameters;
							// Set status output that update is done
							UpdateDone															:= TRUE;
						ELSE
							// PARAMTERS ARE INVALID
							IF (Parameters.ParameterNumber = 0) THEN
								Internal.AddErrorInfo											:= 'Parameter ID is invalid';
							ELSIF (Parameters.SectionID > HMI_CONFIG_NR_OF_SECTIONS) THEN
								Internal.AddErrorInfo											:= 'Number of section is invalid';
							END_IF;
							Internal.ArEventLogWrite.EventID									:= HMI_ERR_WRONG_PARAMETER;
							// Write logbook entry
							WriteLogbookEntry;
							// Set error
							StatusID															:= HMI_ERR_WRONG_PARAMETER;
							Error																:= TRUE;
						END_IF;
					ELSIF NOT Update THEN
						UpdateDone																:= FALSE;
					END_IF;

					//:::::::::::::::::::::::::::::::::::::::::::::::::::::::::::::::::::::::::::://
					// Service Channel implementation
					// Check if paramter should be written
					IF ReadUDINT AND NOT(CommandDone) THEN
						// Check if parameters are valid
						IF (Parameters.ParameterNumber <> 0) AND
							(Parameters.SectionID <= HMI_CONFIG_NR_OF_SECTIONS) THEN
							// PARAMTERS ARE VALID
							// copy paramters to internal stucture
							Internal.ParametersUsed												:= Parameters;
							Internal.Status.ReadStatus := SuperTrakServChanRead(Parameters.SectionID,Parameters.ParameterNumber,Parameters.StartParameterIndex,Parameters.ParameterValueCount,ADR(Out_UDINT),SIZEOF(Out_UDINT));
							IF Internal.Status.ReadStatus <> 0 THEN
								Internal.AddErrorInfo											:= 'Command was not executed successfully: ';
								Info.ErrorCode													:= Internal.Status.ReadStatus;
								GetErrorCode;
								Internal.ArEventLogWrite.EventID								:= HMI_ERR_CMD_NOT_EXECUTED;
								// Write logbook entry
								WriteLogbookEntry;
								// Set error
								StatusID														:= HMI_ERR_CMD_NOT_EXECUTED;
								Error															:= TRUE;
							ELSE
								CommandDone														:= TRUE;
							END_IF;
						ELSE
							// PARAMTERS ARE INVALID
							IF (Parameters.ParameterNumber = 0) THEN
								Internal.AddErrorInfo											:= 'Parameter ID is invalid';
							ELSIF (Parameters.SectionID > HMI_CONFIG_NR_OF_SECTIONS) THEN
								Internal.AddErrorInfo											:= 'Number of section is invalid';
							END_IF;
							Internal.ArEventLogWrite.EventID									:= HMI_ERR_WRONG_PARAMETER;
							// Write logbook entry
							WriteLogbookEntry;
							// Set error
							StatusID															:= HMI_ERR_WRONG_PARAMETER;
							Error																:= TRUE;
						END_IF;

					ELSIF ReadUINT AND NOT(CommandDone) THEN
						// Check if parameters are valid
						IF (Parameters.ParameterNumber <> 0) AND
							(Parameters.SectionID <= HMI_CONFIG_NR_OF_SECTIONS) THEN
							// PARAMTERS ARE VALID
							// copy paramters to internal stucture
							Internal.ParametersUsed												:= Parameters;
							Internal.Status.ReadStatus := SuperTrakServChanRead(Parameters.SectionID,Parameters.ParameterNumber,Parameters.StartParameterIndex,Parameters.ParameterValueCount,ADR(Out_UINT),SIZEOF(Out_UINT));
							IF Internal.Status.ReadStatus <> 0 THEN
								Internal.AddErrorInfo											:= 'Command was not executed successfully: ';
								Info.ErrorCode													:= Internal.Status.ReadStatus;
								GetErrorCode;
								Internal.ArEventLogWrite.EventID								:= HMI_ERR_CMD_NOT_EXECUTED;
								// Write logbook entry
								WriteLogbookEntry;
								// Set error
								StatusID														:= HMI_ERR_CMD_NOT_EXECUTED;
								Error															:= TRUE;
							ELSE
								CommandDone														:= TRUE;
							END_IF;
						ELSE
							// PARAMTERS ARE INVALID
							IF (Parameters.ParameterNumber = 0) THEN
								Internal.AddErrorInfo											:= 'Parameter ID is invalid';
							ELSIF (Parameters.SectionID > HMI_CONFIG_NR_OF_SECTIONS) THEN
								Internal.AddErrorInfo											:= 'Number of section is invalid';
							END_IF;
							Internal.ArEventLogWrite.EventID									:= HMI_ERR_WRONG_PARAMETER;
							// Write logbook entry
							WriteLogbookEntry;
							// Set error
							StatusID															:= HMI_ERR_WRONG_PARAMETER;
							Error																:= TRUE;
						END_IF;

					ELSIF ReadUSINT AND NOT(CommandDone) THEN
						// Check if parameters are valid
						IF (Parameters.ParameterNumber <> 0) AND
							(Parameters.SectionID <= HMI_CONFIG_NR_OF_SECTIONS) THEN
							// PARAMTERS ARE VALID
							// copy paramters to internal stucture
							Internal.ParametersUsed												:= Parameters;
							Internal.Status.ReadStatus := SuperTrakServChanRead(Parameters.SectionID,Parameters.ParameterNumber,Parameters.StartParameterIndex,Parameters.ParameterValueCount,ADR(Out_USINT),SIZEOF(Out_USINT));
							IF Internal.Status.ReadStatus <> 0 THEN
								Internal.AddErrorInfo											:= 'Command was not executed successfully: ';
								Info.ErrorCode													:= Internal.Status.ReadStatus;
								GetErrorCode;
								Internal.ArEventLogWrite.EventID								:= HMI_ERR_CMD_NOT_EXECUTED;
								// Write logbook entry
								WriteLogbookEntry;
								// Set error
								StatusID														:= HMI_ERR_CMD_NOT_EXECUTED;
								Error															:= TRUE;
							ELSE
								CommandDone														:= TRUE;
							END_IF;
						ELSE
							// PARAMTERS ARE INVALID
							IF (Parameters.ParameterNumber = 0) THEN
								Internal.AddErrorInfo											:= 'Parameter ID is invalid';
							ELSIF (Parameters.SectionID > HMI_CONFIG_NR_OF_SECTIONS) THEN
								Internal.AddErrorInfo											:= 'Number of section is invalid';
							END_IF;
							Internal.ArEventLogWrite.EventID									:= HMI_ERR_WRONG_PARAMETER;
							// Write logbook entry
							WriteLogbookEntry;
							// Set error
							StatusID															:= HMI_ERR_WRONG_PARAMETER;
							Error																:= TRUE;
						END_IF;

					ELSIF ReadDINT AND NOT(CommandDone) THEN
						// Check if parameters are valid
						IF (Parameters.ParameterNumber <> 0) AND
							(Parameters.SectionID <= HMI_CONFIG_NR_OF_SECTIONS) THEN
							// PARAMTERS ARE VALID
							// copy paramters to internal stucture
							Internal.ParametersUsed												:= Parameters;
							Internal.Status.ReadStatus := SuperTrakServChanRead(Parameters.SectionID,Parameters.ParameterNumber,Parameters.StartParameterIndex,Parameters.ParameterValueCount,ADR(Out_DINT),SIZEOF(Out_DINT));
							IF Internal.Status.ReadStatus <> 0 THEN
								Internal.AddErrorInfo											:= 'Command was not executed successfully: ';
								Info.ErrorCode													:= Internal.Status.ReadStatus;
								GetErrorCode;
								Internal.ArEventLogWrite.EventID								:= HMI_ERR_CMD_NOT_EXECUTED;
								// Write logbook entry
								WriteLogbookEntry;
								// Set error
								StatusID														:= HMI_ERR_CMD_NOT_EXECUTED;
								Error															:= TRUE;
							ELSE
								CommandDone														:= TRUE;
							END_IF;
						ELSE
							// PARAMTERS ARE INVALID
							IF (Parameters.ParameterNumber = 0) THEN
								Internal.AddErrorInfo											:= 'Parameter ID is invalid';
							ELSIF (Parameters.SectionID > HMI_CONFIG_NR_OF_SECTIONS) THEN
								Internal.AddErrorInfo											:= 'Number of section is invalid';
							END_IF;
							Internal.ArEventLogWrite.EventID									:= HMI_ERR_WRONG_PARAMETER;
							// Write logbook entry
							WriteLogbookEntry;
							// Set error
							StatusID															:= HMI_ERR_WRONG_PARAMETER;
							Error																:= TRUE;
						END_IF;

					ELSIF ReadINT AND NOT(CommandDone) THEN
						// Check if parameters are valid
						IF (Parameters.ParameterNumber <> 0) AND
							(Parameters.SectionID <= HMI_CONFIG_NR_OF_SECTIONS) THEN
							// PARAMTERS ARE VALID
							// copy paramters to internal stucture
							Internal.ParametersUsed												:= Parameters;
							Internal.Status.ReadStatus := SuperTrakServChanRead(Parameters.SectionID,Parameters.ParameterNumber,Parameters.StartParameterIndex,Parameters.ParameterValueCount,ADR(Out_INT),SIZEOF(Out_INT));
							IF Internal.Status.ReadStatus <> 0 THEN
								Internal.AddErrorInfo											:= 'Command was not executed successfully: ';
								Info.ErrorCode													:= Internal.Status.ReadStatus;
								GetErrorCode;
								Internal.ArEventLogWrite.EventID								:= HMI_ERR_CMD_NOT_EXECUTED;
								// Write logbook entry
								WriteLogbookEntry;
								// Set error
								StatusID														:= HMI_ERR_CMD_NOT_EXECUTED;
								Error															:= TRUE;
							ELSE
								CommandDone														:= TRUE;
							END_IF;
						ELSE
							// PARAMTERS ARE INVALID
							IF (Parameters.ParameterNumber = 0) THEN
								Internal.AddErrorInfo											:= 'Parameter ID is invalid';
							ELSIF (Parameters.SectionID > HMI_CONFIG_NR_OF_SECTIONS) THEN
								Internal.AddErrorInfo											:= 'Number of section is invalid';
							END_IF;
							Internal.ArEventLogWrite.EventID									:= HMI_ERR_WRONG_PARAMETER;
							// Write logbook entry
							WriteLogbookEntry;
							// Set error
							StatusID															:= HMI_ERR_WRONG_PARAMETER;
							Error																:= TRUE;
						END_IF;

					ELSIF ReadSINT AND NOT(CommandDone) THEN
						// Check if parameters are valid
						IF (Parameters.ParameterNumber <> 0) AND
							(Parameters.SectionID <= HMI_CONFIG_NR_OF_SECTIONS) THEN
							// PARAMTERS ARE VALID
							// copy paramters to internal stucture
							Internal.ParametersUsed												:= Parameters;
							Internal.Status.ReadStatus := SuperTrakServChanRead(Parameters.SectionID,Parameters.ParameterNumber,Parameters.StartParameterIndex,Parameters.ParameterValueCount,ADR(Out_SINT),SIZEOF(Out_SINT));
							IF Internal.Status.ReadStatus <> 0 THEN
								Internal.AddErrorInfo											:= 'Command was not executed successfully: ';
								Info.ErrorCode													:= Internal.Status.ReadStatus;
								GetErrorCode;
								Internal.ArEventLogWrite.EventID								:= HMI_ERR_CMD_NOT_EXECUTED;
								// Write logbook entry
								WriteLogbookEntry;
								// Set error
								StatusID														:= HMI_ERR_CMD_NOT_EXECUTED;
								Error															:= TRUE;
							ELSE
								CommandDone														:= TRUE;
							END_IF;
						ELSE
							// PARAMTERS ARE INVALID
							IF (Parameters.ParameterNumber = 0) THEN
								Internal.AddErrorInfo											:= 'Parameter ID is invalid';
							ELSIF (Parameters.SectionID > HMI_CONFIG_NR_OF_SECTIONS) THEN
								Internal.AddErrorInfo											:= 'Number of section is invalid';
							END_IF;
							Internal.ArEventLogWrite.EventID									:= HMI_ERR_WRONG_PARAMETER;
							// Write logbook entry
							WriteLogbookEntry;
							// Set error
							StatusID															:= HMI_ERR_WRONG_PARAMETER;
							Error																:= TRUE;
						END_IF;

					ELSIF ReadREAL AND NOT(CommandDone) THEN
						// Check if parameters are valid
						IF (Parameters.ParameterNumber <> 0) AND
							(Parameters.SectionID <= HMI_CONFIG_NR_OF_SECTIONS) THEN
							// PARAMTERS ARE VALID
							// copy paramters to internal stucture
							Internal.ParametersUsed												:= Parameters;
							Internal.Status.ReadStatus := SuperTrakServChanRead(Parameters.SectionID,Parameters.ParameterNumber,Parameters.StartParameterIndex,Parameters.ParameterValueCount,ADR(Out_REAL),SIZEOF(Out_REAL));
							IF Internal.Status.ReadStatus <> 0 THEN
								Internal.AddErrorInfo											:= 'Command was not executed successfully: ';
								Info.ErrorCode													:= Internal.Status.ReadStatus;
								GetErrorCode;
								Internal.ArEventLogWrite.EventID								:= HMI_ERR_CMD_NOT_EXECUTED;
								// Write logbook entry
								WriteLogbookEntry;
								// Set error
								StatusID														:= HMI_ERR_CMD_NOT_EXECUTED;
								Error															:= TRUE;
							ELSE
								CommandDone														:= TRUE;
							END_IF;
						ELSE
							// PARAMTERS ARE INVALID
							IF (Parameters.ParameterNumber = 0) THEN
								Internal.AddErrorInfo											:= 'Parameter ID is invalid';
							ELSIF (Parameters.SectionID > HMI_CONFIG_NR_OF_SECTIONS) THEN
								Internal.AddErrorInfo											:= 'Number of section is invalid';
							END_IF;
							Internal.ArEventLogWrite.EventID									:= HMI_ERR_WRONG_PARAMETER;
							// Write logbook entry
							WriteLogbookEntry;
							// Set error
							StatusID															:= HMI_ERR_WRONG_PARAMETER;
							Error																:= TRUE;
						END_IF;

					ELSIF ReadSTRING AND NOT(CommandDone) THEN
						// Check if parameters are valid
						IF (Parameters.ParameterNumber <> 0) AND
							(Parameters.SectionID <= HMI_CONFIG_NR_OF_SECTIONS) AND
							(Parameters.STRINGsize > 0) THEN
							// PARAMTERS ARE VALID
							// copy paramters to internal stucture
							Internal.ParametersUsed												:= Parameters;
							Internal.Status.ReadStatus := SuperTrakServChanRead(Parameters.SectionID,Parameters.ParameterNumber,Parameters.StartParameterIndex,Parameters.STRINGsize,ADR(Out_STRING),Parameters.STRINGsize);
							IF Internal.Status.ReadStatus <> 0 THEN
								Internal.AddErrorInfo											:= 'Command was not executed successfully: ';
								Info.ErrorCode													:= Internal.Status.ReadStatus;
								GetErrorCode;
								Internal.ArEventLogWrite.EventID								:= HMI_ERR_CMD_NOT_EXECUTED;
								// Write logbook entry
								WriteLogbookEntry;
								// Set error
								StatusID														:= HMI_ERR_CMD_NOT_EXECUTED;
								Error															:= TRUE;
							ELSE
								CommandDone														:= TRUE;
							END_IF;
						ELSE
							// PARAMTERS ARE INVALID
							IF (Parameters.ParameterNumber = 0) THEN
								Internal.AddErrorInfo											:= 'Parameter ID is invalid';
							ELSIF (Parameters.SectionID > HMI_CONFIG_NR_OF_SECTIONS) THEN
								Internal.AddErrorInfo											:= 'Number of section is invalid';
							END_IF;
							Internal.ArEventLogWrite.EventID									:= HMI_ERR_WRONG_PARAMETER;
							// Write logbook entry
							WriteLogbookEntry;
							// Set error
							StatusID															:= HMI_ERR_WRONG_PARAMETER;
							Error																:= TRUE;
						END_IF;
					END_IF;

					IF NOT(ReadUDINT) AND NOT(ReadUINT) AND NOT(ReadUSINT) AND NOT(ReadDINT) AND NOT(ReadINT) AND NOT(ReadSINT) AND NOT(ReadREAL) AND NOT(ReadSTRING) THEN
						CommandDone	:= FALSE;
					END_IF;

					//:::::::::::::::::::::::::::::::::::::::::::::::::::::::::::::::::::::::::::://
					// Error detection
					// Check if communication is not established
					IF NOT HMILink.SuperTrakStatus.StatusValid THEN
						IF (HMILink.LibraryStatus.FbID[0] = 0) AND (HMILink.LibraryStatus.LogBookIdent <> 0) THEN
							Internal.AddErrorInfo												:= 'No enabled instance of HMIControl could be found';
							Internal.ArEventLogWrite.EventID									:= HMI_ERR_NO_HMICONTROL_REG;
							// Write logbook entry
							WriteLogbookEntry;
							// Set error
							StatusID															:= HMI_ERR_NO_HMICONTROL_REG;
							Error																:= TRUE;
						ELSE
							// Set error
							Internal.AddErrorInfo												:= 'No communication to SuperTrak';
							Internal.ArEventLogWrite.EventID									:= HMI_ERR_COMMUNICAITON_TIME_OUT;
							// Write logbook entry
							WriteLogbookEntry;
							StatusID															:= HMI_ERR_COMMUNICAITON_TIME_OUT;
							Error																:= TRUE;
						END_IF;
					END_IF;
				ELSE
					Internal.Status.InitConfigCheckDone											:= FALSE;
					// Set error
					StatusID																	:= HMI_ERR_WRONG_CONFIG;
					Error																		:= TRUE;
				END_IF;

				//--------------------------------------------------------------------------------//
				// Error handling
				//--------------------------------------------------------------------------------//
			HMI_RPAR_STATE_ERROR:

				// Reset active output
				Active																		:= FALSE;

				UpdateDone																	:= FALSE;
				CommandDone																	:= FALSE;

				IF NOT Error THEN
					// Check in which state to jump
					IF NOT Internal.Status.FuncitonBlockRegistered THEN
						Internal.Step														:= HMI_RPAR_STATE_INIT;
					ELSIF NOT Internal.Status.InitConfigCheckDone THEN
						Internal.Step														:= HMI_RPAR_STATE_INIT;
					ELSIF NOT Internal.Status.InitParCheckDone THEN
						Internal.Step														:= HMI_RPAR_STATE_INIT_CHECK_PAR;
					ELSE
						Internal.Step														:= HMI_RPAR_STATE_OPERATION;
					END_IF;
				END_IF;

		END_CASE;

		//************************************************************************************//
		// Error and Warning acknowledgement
		//************************************************************************************//

		// Check if error or warning is acknowledged by user
		IF ErrorReset AND Error AND NOT Internal.ErrorResetOld THEN
			// Reset error
			StatusID																		:= HMI_NO_ERROR;
			Error																			:= FALSE;
			Internal.Status.ReadStatus														:= 0;
			Info.ErrorCode																	:= 0;
		ELSIF ErrorReset AND StatusID <> HMI_NO_ERROR AND NOT Internal.ErrorResetOld THEN
			// Reset warning
			StatusID																		:= HMI_NO_ERROR;
			Internal.Status.ReadStatus														:= 0;
			Info.ErrorCode																	:= 0;
		END_IF;

		// Copy command for edge detection
		Internal.ErrorResetOld																:= ErrorReset;
		Internal.UpdateOld																	:= Update;

	ELSE
		//####################################################################################//
		// FUNCTION BLOCK IS DISABLED
		//####################################################################################//
		// Reset all outputs
		Active																				:= FALSE;
		Error																				:= FALSE;
		StatusID																			:= 0;
		UpdateDone																			:= FALSE;

		CommandDone																			:= FALSE;

		Internal.Status.FuncitonBlockRegistered												:= FALSE;
		Internal.Status.InitParCheckDone													:= FALSE;
		Internal.Status.InitConfigCheckDone													:= FALSE;
		Internal.Step																		:= HMI_RPAR_STATE_INIT;

		Internal.Status.ReadStatus															:= 0;
		Info.ErrorCode																		:= 0;
	END_IF;
END_FUNCTION_BLOCK
```
